// TIA Portal V17 export
// export: Created 2023-04-11T09:33:36.8742069Z, ExportSetting WithDefaults, DisplayName Totally Integrated Automation Portal, DisplayVersion V17 Update 3, DisplayName TIA Portal Openness, DisplayVersion V17 Update 3, DisplayName TIA Portal Version Control Interface, DisplayVersion V17, DisplayName SINAMICS Startdrive Advanced, DisplayVersion V17 Update2, DisplayName SINAMICS Startdrive G130, G150, S120, S150, SINAMICS MV, S210, DisplayVersion V17 Update2, DisplayName SINAMICS Startdrive G110M, G120, G120C, G120D, G120P, G115D, DisplayVersion V17 Update2, DisplayName STEP 7 Professional, DisplayVersion V17 Update 3, DisplayName STEP 7 Safety, DisplayVersion V17, DisplayName WinCC UA Professional, DisplayVersion V17 Update 3
FUNCTION_BLOCK "FB_dTag"   // FB110, LAD
{ S7_Optimized_Access := 'TRUE' }
VERSION : 0.1
// stored: AutoNumber true, IsIECCheckEnabled false, IsRetainMemResEnabled false, MemoryReserve 100, SetENOAutomatically false, UDAEnableTagReadback false
   VAR_INPUT
      trigRead : Bool;
      projetWrite : DInt;
      versionWrite : Int;
      x_BitData : Bool;
   END_VAR
   VAR_OUTPUT
      readData_ok : Bool;
      readData_err : Bool;
      projectRead : DInt;
      versionRead : Int;
      writeDataDone : Bool;
      y_BitData : Bool;
      y_bitClk : Bool;
   END_VAR
   VAR_IN_OUT
      trigWrite_io : Bool;
   END_VAR
   VAR
      w_data : Array[0..2] of Int;
      r_data : Array[0..2] of Int;
      readingActive : Bool;
      writingActive : Bool;
      writeInit : Bool;
      clk_lo : Bool;
      clk_hi : Bool;
      readStrobe : Bool;
      writeStrobe : Bool;
      readDataReady : Bool;
      ready : Bool;
      currReadBit : Int;
      currWriteBit : Int;
      readDataArr : Array[0..39] of Bool;
      writeDataArr : Array[0..71] of Bool;
      IEC_Timer_0_Instance_1 { S7_SetPoint := 'True'} : TON_TIME;
      IEC_Timer_0_Instance { S7_SetPoint := 'True'} : TON_TIME;
      IEC_Timer_0_Instance_2 { S7_SetPoint := 'True'} : TON_TIME;
      edge : Array[0..2] of Bool;
      IEC_Timer_0_Instance_3 { S7_SetPoint := 'True'} : TON_TIME;
      IEC_Timer_0_Instance_4 { S7_SetPoint := 'True'} : TON_TIME;
      IEC_Timer_0_Instance_5 { S7_SetPoint := 'True'} : TON_TIME;
      lrc { ExternalAccessible := 'False'; ExternalVisible := 'False'; ExternalWritable := 'False'} : Int;
   END_VAR
   VAR_TEMP
      tempIndex : Int;
   END_VAR
   VAR_TEMP   // added for the SCL form of the ladder/FBD networks
      _w1 : Bool;
      _w2 : Bool;
      _w3 : Bool;
   END_VAR
BEGIN

REGION Network 1 (SCL): Prepare write / multiplex read data
   // Prepare write data
   IF #trigWrite_io THEN
       //
       #w_data[0] := #projetWrite.%W0;
       #w_data[1] := #projetWrite.%W1;
       #w_data[1] := #w_data[1] AND 16#07FF;

       // temp_buffer
       #w_data[1] := #w_data[1] OR SHL(IN := (#versionWrite AND 16#1F), N := 11);

   END_IF;

   // Multiplex read data
   #projectRead.%W0 := #r_data[0];
   #projectRead.%W1 := #r_data[1] AND 16#07FF;
   #versionRead := SHR(IN := (#r_data[1] AND 16#F800), N := 11);
END_REGION

REGION Network 3: Idle
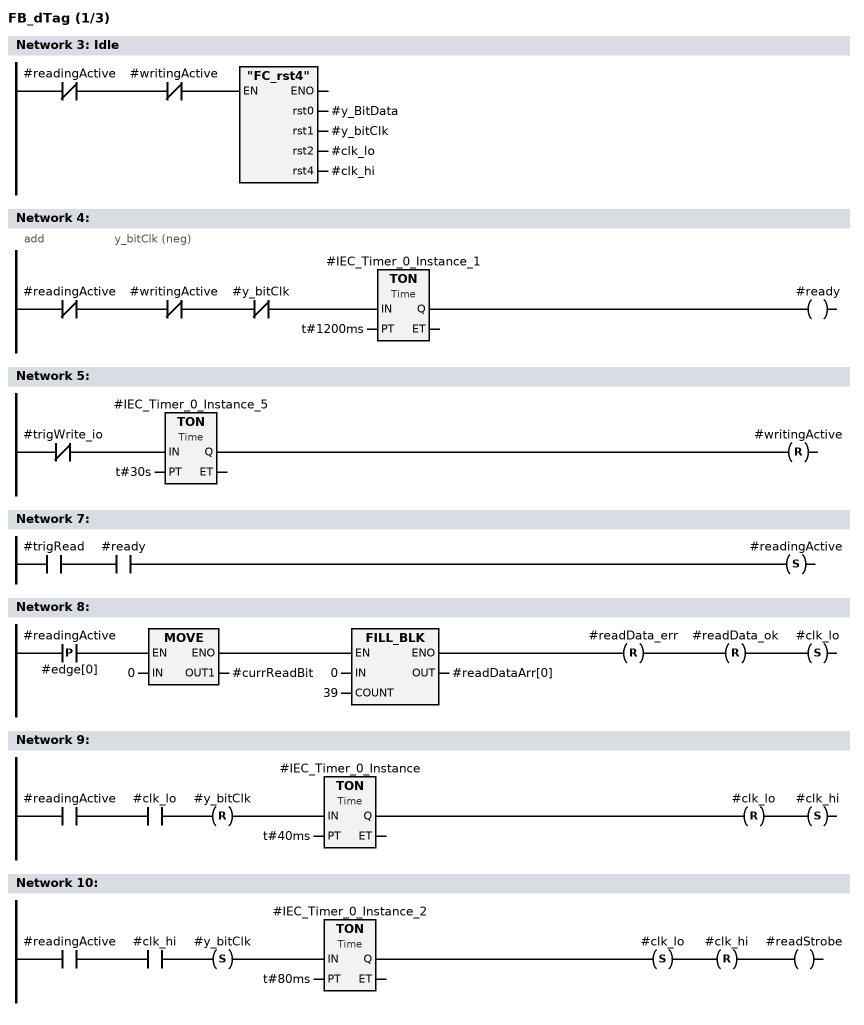
   RUNG wire#powerrail
      I_Contact( #readingActive )
      I_Contact( #writingActive )
      "FC_rst4"(rst0 => #y_BitData, rst1 => #y_bitClk, rst2 => #clk_lo, rst4 => #clk_hi)
   END_RUNG
   // the same network as SCL:
   IF NOT #readingActive AND NOT #writingActive THEN
       "FC_rst4"(rst0 => #y_BitData, rst1 => #y_bitClk, rst2 => #clk_lo, rst4 => #clk_hi);
   END_IF;
END_REGION

REGION Network 4
   // add                    y_bitClk (neg)
   RUNG wire#powerrail
      I_Contact( #readingActive )
      I_Contact( #writingActive )
      I_Contact( #y_bitClk )
      { S7_Templates := "time_type := Time" } #IEC_Timer_0_Instance_1.TON(pt := t#1200ms, et =>)
      Coil( #ready )
   END_RUNG
   // the same network as SCL:
   #IEC_Timer_0_Instance_1(IN := NOT #readingActive AND NOT #writingActive AND NOT #y_bitClk, PT := t#1200ms);   // TON
   #ready := #IEC_Timer_0_Instance_1.Q;
END_REGION

REGION Network 5
   RUNG wire#powerrail
      I_Contact( #trigWrite_io )
      { S7_Templates := "time_type := Time" } #IEC_Timer_0_Instance_5.TON(pt := t#30s, et =>)
      R_Coil( #writingActive )
   END_RUNG
   // the same network as SCL:
   #IEC_Timer_0_Instance_5(IN := NOT #trigWrite_io, PT := t#30s);   // TON
   IF #IEC_Timer_0_Instance_5.Q THEN #writingActive := FALSE; END_IF;
END_REGION

REGION Network 6: --------- Reading ------------
END_REGION

REGION Network 7
   RUNG wire#powerrail
      Contact( #trigRead )
      Contact( #ready )
      S_Coil( #readingActive )
   END_RUNG
   // the same network as SCL:
   IF #trigRead AND #ready THEN #readingActive := TRUE; END_IF;
END_REGION

REGION Network 8
   RUNG wire#powerrail
      P_Contact(operand := #readingActive, bit := #edge[0])
      Move(in := 0, out1 => #currReadBit)
      FillBlockI(in := 0, count := 39, out => #readDataArr[0])
      R_Coil( #readData_err )
      R_Coil( #readData_ok )
      S_Coil( #clk_lo )
   END_RUNG
   // the same network as SCL:
   #_w1 := #readingActive AND NOT #edge[0];   // rising edge of #readingActive
   #edge[0] := #readingActive;
   IF #_w1 THEN
       #currReadBit := 0;
       FILL_BLK(IN := 0, COUNT := 39, OUT => #readDataArr[0]);
       #readData_err := FALSE;
       #readData_ok := FALSE;
       #clk_lo := TRUE;
   END_IF;
END_REGION

REGION Network 9
   RUNG wire#powerrail
      Contact( #readingActive )
      Contact( #clk_lo )
      R_Coil( #y_bitClk )
      { S7_Templates := "time_type := Time" } #IEC_Timer_0_Instance.TON(pt := t#40ms, et =>)
      R_Coil( #clk_lo )
      S_Coil( #clk_hi )
   END_RUNG
   // the same network as SCL:
   #_w1 := #readingActive AND #clk_lo;
   IF #_w1 THEN #y_bitClk := FALSE; END_IF;
   #IEC_Timer_0_Instance(IN := #_w1, PT := t#40ms);   // TON
   IF #IEC_Timer_0_Instance.Q THEN
       #clk_lo := FALSE;
       #clk_hi := TRUE;
   END_IF;
END_REGION

REGION Network 10
   RUNG wire#powerrail
      Contact( #readingActive )
      Contact( #clk_hi )
      S_Coil( #y_bitClk )
      { S7_Templates := "time_type := Time" } #IEC_Timer_0_Instance_2.TON(pt := t#80ms, et =>)
      S_Coil( #clk_lo )
      R_Coil( #clk_hi )
      Coil( #readStrobe )
   END_RUNG
   // the same network as SCL:
   #_w1 := #readingActive AND #clk_hi;
   IF #_w1 THEN #y_bitClk := TRUE; END_IF;
   #IEC_Timer_0_Instance_2(IN := #_w1, PT := t#80ms);   // TON
   IF #IEC_Timer_0_Instance_2.Q THEN
       #clk_lo := TRUE;
       #clk_hi := FALSE;
   END_IF;
   #readStrobe := #IEC_Timer_0_Instance_2.Q;
END_REGION

REGION Network 11
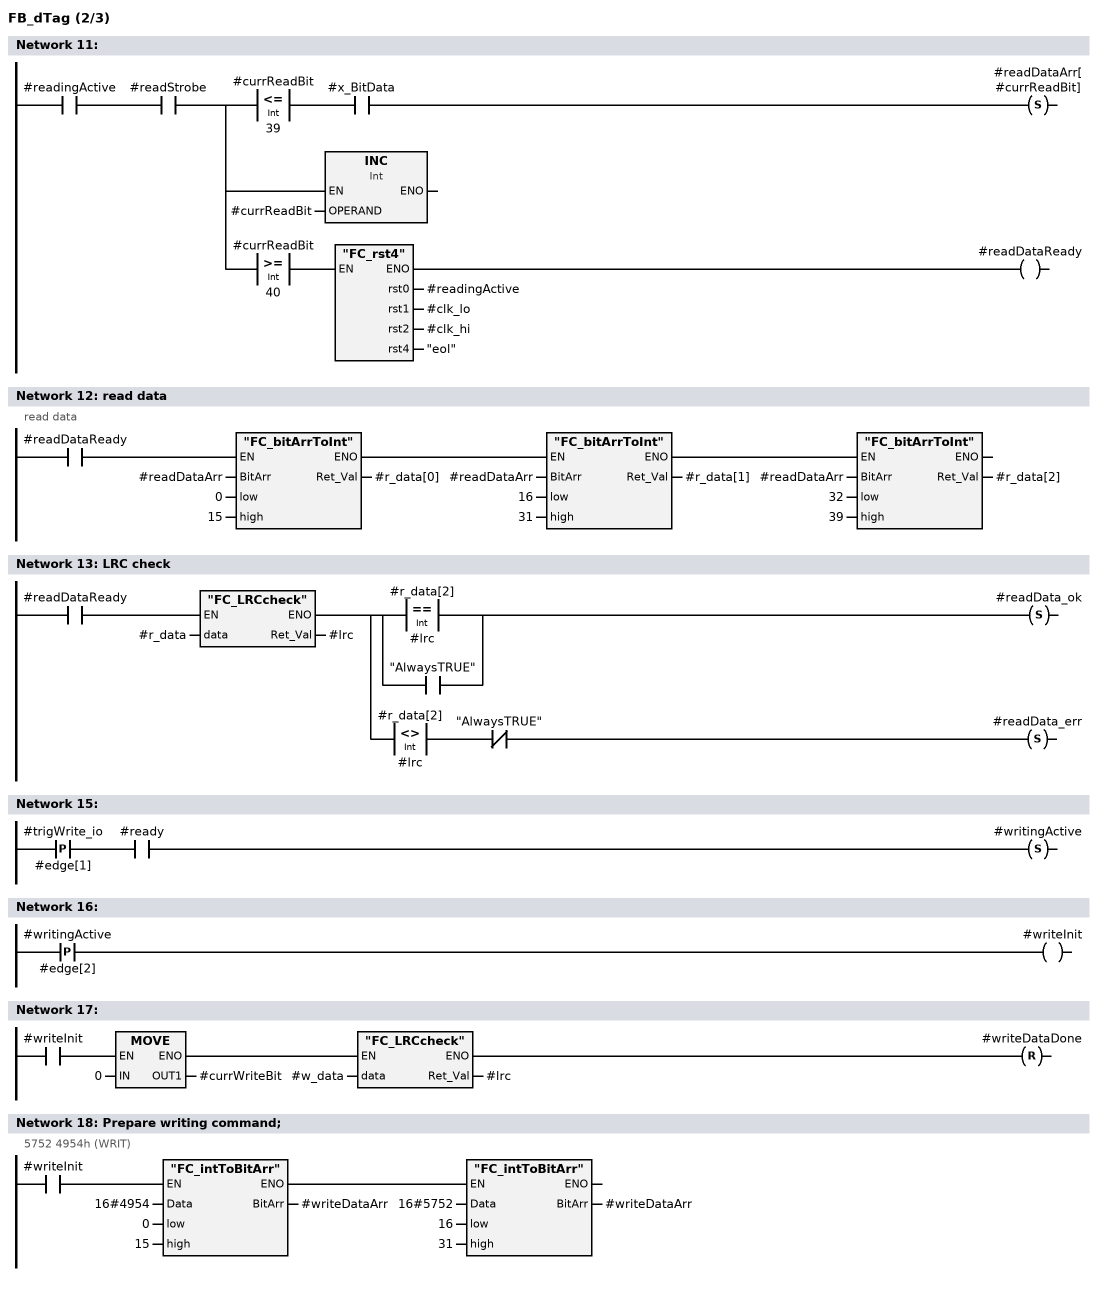
   RUNG wire#powerrail
      Contact( #readingActive )
      Contact( #readStrobe )
      wire#w1
      { S7_Templates := "SrcType := Int" } LE_Contact(in1 := #currReadBit, in2 := 39)
      Contact( #x_BitData )
      S_Coil( #readDataArr[#currReadBit] )
   END_RUNG
   RUNG wire#w1
      { S7_Templates := "DestType := Int" } Inc( #currReadBit )
   END_RUNG
   RUNG wire#w1
      { S7_Templates := "SrcType := Int" } GE_Contact(in1 := #currReadBit, in2 := 40)
      "FC_rst4"(rst0 => #readingActive, rst1 => #clk_lo, rst2 => #clk_hi, rst4 => "eol")
      Coil( #readDataReady )
   END_RUNG
   // the same network as SCL:
   #_w1 := #readingActive AND #readStrobe;
   IF #_w1 AND (#currReadBit <= 39) AND #x_BitData THEN #readDataArr[#currReadBit] := TRUE; END_IF;
   IF #_w1 THEN #currReadBit := #currReadBit + 1; END_IF;
   "FC_rst4"(EN := #_w1 AND (#currReadBit >= 40),
             rst0 => #readingActive,
             rst1 => #clk_lo,
             rst2 => #clk_hi,
             rst4 => "eol",
             ENO => #_w2);
   #readDataReady := #_w2;
END_REGION

REGION Network 12: read data
   // read data
   RUNG wire#powerrail
      Contact( #readDataReady )
      "FC_bitArrToInt"(BitArr := #readDataArr, low := 0, high := 15, Ret_Val => #r_data[0])
      "FC_bitArrToInt"(BitArr := #readDataArr, low := 16, high := 31, Ret_Val => #r_data[1])
      "FC_bitArrToInt"(BitArr := #readDataArr, low := 32, high := 39, Ret_Val => #r_data[2])
   END_RUNG
   // the same network as SCL:
   #r_data[0] := "FC_bitArrToInt"(EN := #readDataReady,
                           BitArr := #readDataArr,
                           low := 0,
                           high := 15,
                           ENO => #_w1);
   #r_data[1] := "FC_bitArrToInt"(EN := #_w1, BitArr := #readDataArr, low := 16, high := 31, ENO => #_w2);
   IF #_w2 THEN #r_data[2] := "FC_bitArrToInt"(BitArr := #readDataArr, low := 32, high := 39); END_IF;
END_REGION

REGION Network 13: LRC check
   RUNG wire#powerrail
      Contact( #readDataReady )
      "FC_LRCcheck"(data := #r_data, Ret_Val => #lrc)
      wire#w1
      { S7_Templates := "SrcType := Int" } EQ_Contact(in1 := #r_data[2], in2 := #lrc)
      wire#w2
      S_Coil( #readData_ok )
   END_RUNG
   RUNG wire#w1
      Contact( "AlwaysTRUE" )
   END_RUNG wire#w2
   RUNG wire#w1
      { S7_Templates := "SrcType := Int" } NE_Contact(in1 := #r_data[2], in2 := #lrc)
      I_Contact( "AlwaysTRUE" )
      S_Coil( #readData_err )
   END_RUNG
   // the same network as SCL:
   #lrc := "FC_LRCcheck"(EN := #readDataReady, data := #r_data, ENO => #_w1);
   IF #_w1 AND ((#r_data[2] = #lrc) OR "AlwaysTRUE") THEN #readData_ok := TRUE; END_IF;
   IF #_w1 AND (#r_data[2] <> #lrc) AND NOT "AlwaysTRUE" THEN #readData_err := TRUE; END_IF;
END_REGION

REGION Network 14: --------- Writing ------------
END_REGION

REGION Network 15
   RUNG wire#powerrail
      P_Contact(operand := #trigWrite_io, bit := #edge[1])
      Contact( #ready )
      S_Coil( #writingActive )
   END_RUNG
   // the same network as SCL:
   #_w1 := #trigWrite_io AND NOT #edge[1];   // rising edge of #trigWrite_io
   #edge[1] := #trigWrite_io;
   IF #_w1 AND #ready THEN #writingActive := TRUE; END_IF;
END_REGION

REGION Network 16
   RUNG wire#powerrail
      P_Contact(operand := #writingActive, bit := #edge[2])
      Coil( #writeInit )
   END_RUNG
   // the same network as SCL:
   #_w1 := #writingActive AND NOT #edge[2];   // rising edge of #writingActive
   #edge[2] := #writingActive;
   #writeInit := #_w1;
END_REGION

REGION Network 17
   RUNG wire#powerrail
      Contact( #writeInit )
      Move(in := 0, out1 => #currWriteBit)
      "FC_LRCcheck"(data := #w_data, Ret_Val => #lrc)
      R_Coil( #writeDataDone )
   END_RUNG
   // the same network as SCL:
   IF #writeInit THEN #currWriteBit := 0; END_IF;
   #lrc := "FC_LRCcheck"(EN := #writeInit, data := #w_data, ENO => #_w1);
   IF #_w1 THEN #writeDataDone := FALSE; END_IF;
END_REGION

REGION Network 18: Prepare writing command;
   // 5752 4954h (WRIT)
   RUNG wire#powerrail
      Contact( #writeInit )
      "FC_intToBitArr"(Data := 16#4954, low := 0, high := 15, BitArr => #writeDataArr)
      "FC_intToBitArr"(Data := 16#5752, low := 16, high := 31, BitArr => #writeDataArr)
   END_RUNG
   // the same network as SCL:
   "FC_intToBitArr"(EN := #writeInit,
                    Data := 16#4954,
                    low := 0,
                    high := 15,
                    BitArr => #writeDataArr,
                    ENO => #_w1);
   IF #_w1 THEN "FC_intToBitArr"(Data := 16#5752, low := 16, high := 31, BitArr => #writeDataArr); END_IF;
END_REGION

REGION Network 19: Prepare writing data; 4bytes + CRC
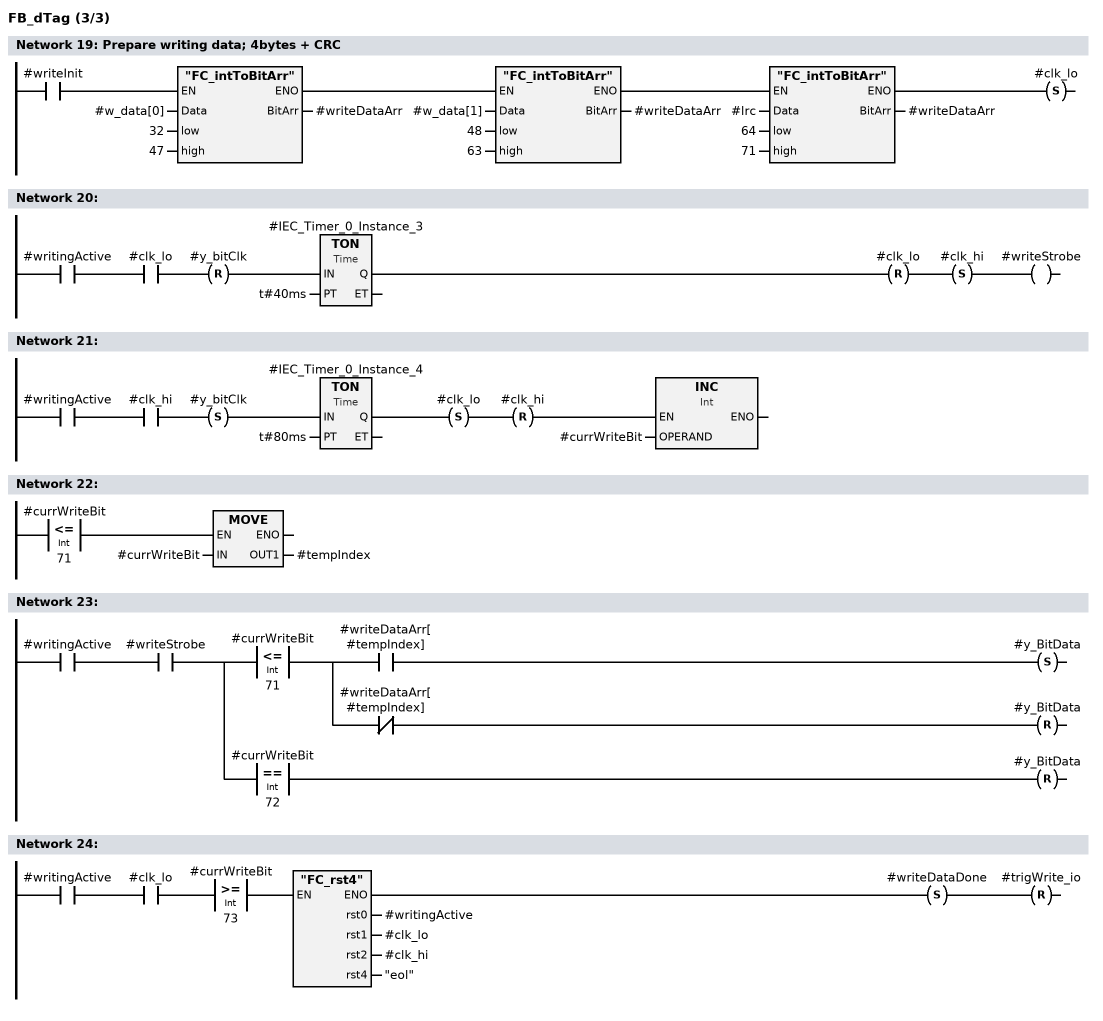
   RUNG wire#powerrail
      Contact( #writeInit )
      "FC_intToBitArr"(Data := #w_data[0], low := 32, high := 47, BitArr => #writeDataArr)
      "FC_intToBitArr"(Data := #w_data[1], low := 48, high := 63, BitArr => #writeDataArr)
      "FC_intToBitArr"(Data := #lrc, low := 64, high := 71, BitArr => #writeDataArr)
      S_Coil( #clk_lo )
   END_RUNG
   // the same network as SCL:
   "FC_intToBitArr"(EN := #writeInit,
                    Data := #w_data[0],
                    low := 32,
                    high := 47,
                    BitArr => #writeDataArr,
                    ENO => #_w1);
   "FC_intToBitArr"(EN := #_w1, Data := #w_data[1], low := 48, high := 63, BitArr => #writeDataArr, ENO => #_w2);
   "FC_intToBitArr"(EN := #_w2, Data := #lrc, low := 64, high := 71, BitArr => #writeDataArr, ENO => #_w3);
   IF #_w3 THEN #clk_lo := TRUE; END_IF;
END_REGION

REGION Network 20
   RUNG wire#powerrail
      Contact( #writingActive )
      Contact( #clk_lo )
      R_Coil( #y_bitClk )
      { S7_Templates := "time_type := Time" } #IEC_Timer_0_Instance_3.TON(pt := t#40ms, et =>)
      R_Coil( #clk_lo )
      S_Coil( #clk_hi )
      Coil( #writeStrobe )
   END_RUNG
   // the same network as SCL:
   #_w1 := #writingActive AND #clk_lo;
   IF #_w1 THEN #y_bitClk := FALSE; END_IF;
   #IEC_Timer_0_Instance_3(IN := #_w1, PT := t#40ms);   // TON
   IF #IEC_Timer_0_Instance_3.Q THEN
       #clk_lo := FALSE;
       #clk_hi := TRUE;
   END_IF;
   #writeStrobe := #IEC_Timer_0_Instance_3.Q;
END_REGION

REGION Network 21
   RUNG wire#powerrail
      Contact( #writingActive )
      Contact( #clk_hi )
      S_Coil( #y_bitClk )
      { S7_Templates := "time_type := Time" } #IEC_Timer_0_Instance_4.TON(pt := t#80ms, et =>)
      S_Coil( #clk_lo )
      R_Coil( #clk_hi )
      { S7_Templates := "DestType := Int" } Inc( #currWriteBit )
   END_RUNG
   // the same network as SCL:
   #_w1 := #writingActive AND #clk_hi;
   IF #_w1 THEN #y_bitClk := TRUE; END_IF;
   #IEC_Timer_0_Instance_4(IN := #_w1, PT := t#80ms);   // TON
   IF #IEC_Timer_0_Instance_4.Q THEN
       #clk_lo := TRUE;
       #clk_hi := FALSE;
       #currWriteBit := #currWriteBit + 1;
   END_IF;
END_REGION

REGION Network 22
   RUNG wire#powerrail
      { S7_Templates := "SrcType := Int" } LE_Contact(in1 := #currWriteBit, in2 := 71)
      Move(in := #currWriteBit, out1 => #tempIndex)
   END_RUNG
   // the same network as SCL:
   IF #currWriteBit <= 71 THEN #tempIndex := #currWriteBit; END_IF;
END_REGION

REGION Network 23
   RUNG wire#powerrail
      Contact( #writingActive )
      Contact( #writeStrobe )
      wire#w1
      { S7_Templates := "SrcType := Int" } LE_Contact(in1 := #currWriteBit, in2 := 71)
      wire#w2
      Contact( #writeDataArr[#tempIndex] )
      S_Coil( #y_BitData )
   END_RUNG
   RUNG wire#w2
      I_Contact( #writeDataArr[#tempIndex] )
      R_Coil( #y_BitData )
   END_RUNG
   RUNG wire#w1
      { S7_Templates := "SrcType := Int" } EQ_Contact(in1 := #currWriteBit, in2 := 72)
      R_Coil( #y_BitData )
   END_RUNG
   // the same network as SCL:
   #_w1 := #writingActive AND #writeStrobe;
   #_w2 := #_w1 AND (#currWriteBit <= 71);
   IF #_w2 AND #writeDataArr[#tempIndex] THEN #y_BitData := TRUE; END_IF;
   IF #_w2 AND NOT #writeDataArr[#tempIndex] THEN #y_BitData := FALSE; END_IF;
   IF #_w1 AND (#currWriteBit = 72) THEN #y_BitData := FALSE; END_IF;
END_REGION

REGION Network 24
   RUNG wire#powerrail
      Contact( #writingActive )
      Contact( #clk_lo )
      { S7_Templates := "SrcType := Int" } GE_Contact(in1 := #currWriteBit, in2 := 73)
      "FC_rst4"(rst0 => #writingActive, rst1 => #clk_lo, rst2 => #clk_hi, rst4 => "eol")
      S_Coil( #writeDataDone )
      R_Coil( #trigWrite_io )
   END_RUNG
   // the same network as SCL:
   "FC_rst4"(EN := #writingActive AND #clk_lo AND (#currWriteBit >= 73),
             rst0 => #writingActive,
             rst1 => #clk_lo,
             rst2 => #clk_hi,
             rst4 => "eol",
             ENO => #_w1);
   IF #_w1 THEN
       #writeDataDone := TRUE;
       #trigWrite_io := FALSE;
   END_IF;
END_REGION
END_FUNCTION_BLOCK
